// TIA Portal V20 export
FUNCTION_BLOCK "CallGlobal"   // FB48, LAD
TITLE = CallGlobal
// All blocks that provide data to the DB Global.Data are called here. That includes blocks to generate system data as well as blocks that connect handle multiple HMIs.
// stored: IsIECCheckEnabled true, MemoryReserve 100, SetENOAutomatically true
   VAR
      statClockSysMemOld { ExternalWritable := 'False'} : Byte;   // Old value system memory evaluation
      statTonTimer : Array[0..10] of IEC_TIMER;
      instLAF_PowerOnOff { ExternalWritable := 'False'} : "LAF_PowerOnOff";
      instLAF_HmiHeaderManager { ExternalWritable := 'False'} : "LAF_HmiHeaderManager";
      instLAF_ClockGen { ExternalWritable := 'False'} : "LAF_ClockGenerator";
      instLSNTP_Server { ExternalWritable := 'False'} : "LSNTP_Server";
      instRemoteAccess { ExternalWritable := 'False'} : "LRemoteAccess_MobilePanelMonitor";
      statPulse : Array[0..99] of Bool;
   END_VAR
   VAR_TEMP
      tempIndex : DInt;   // Temp variable for for loop
      tempAcknowledge : Bool;   // Summarized acknowledge command
      tempPowerOff : Bool;   // Summarized power off command
      tempPowerOn : Bool;   // Summarized power on command
      tempPowerStatus : Int;   // 0 - Off, 1 - Paused, 2 - On
      tempResultXor : Byte;   // Interim result of XOR operation
      tempPosPulse : Byte;   // Interim result puls calculation
   END_VAR
   VAR CONSTANT
      RESET_BUTTON__COULD_BE_ADDED_HERE : Bool := false;   // Placeholder for a potential global reset button
      TRUE : Bool := true;
   END_VAR
   VAR_TEMP   // added for the SCL form of the ladder/FBD networks
      _w1 : Bool;
      _w2 : Bool;
      _w3 : Bool;
   END_VAR
BEGIN

REGION Network 1 (SCL): Summarize HMI commands
   // Read commands for acknowledge, powerOn and powerOff from the different HMI panels and summarize them in temp variables for further logic in this block.
   // Initialize temp variables
   #tempAcknowledge :=
   #tempPowerOff :=
   #tempPowerOn := FALSE;

   // Loop through the HMI panels and summarize the commands
   FOR #tempIndex := 0 TO "NO_OF_PANELS" DO
       #tempAcknowledge := #tempAcknowledge OR "Hmi".mainHeader[#tempIndex].hmiToPlc.acknowledge;
       #tempPowerOff := #tempPowerOff OR "Hmi".mainHeader[#tempIndex].hmiToPlc.powerCommands.%X0;
       #tempPowerOn := #tempPowerOn OR "Hmi".mainHeader[#tempIndex].hmiToPlc.powerCommands.%X1;
   END_FOR;
END_REGION

REGION Network 2: Global Acknowledge
   // The global acknowledge command from the hmi button is assigned to Global.Data.general.acknowledge: This bit it forwarded to all underlaying modules
   // If a hard-wired global reset button exists, it can
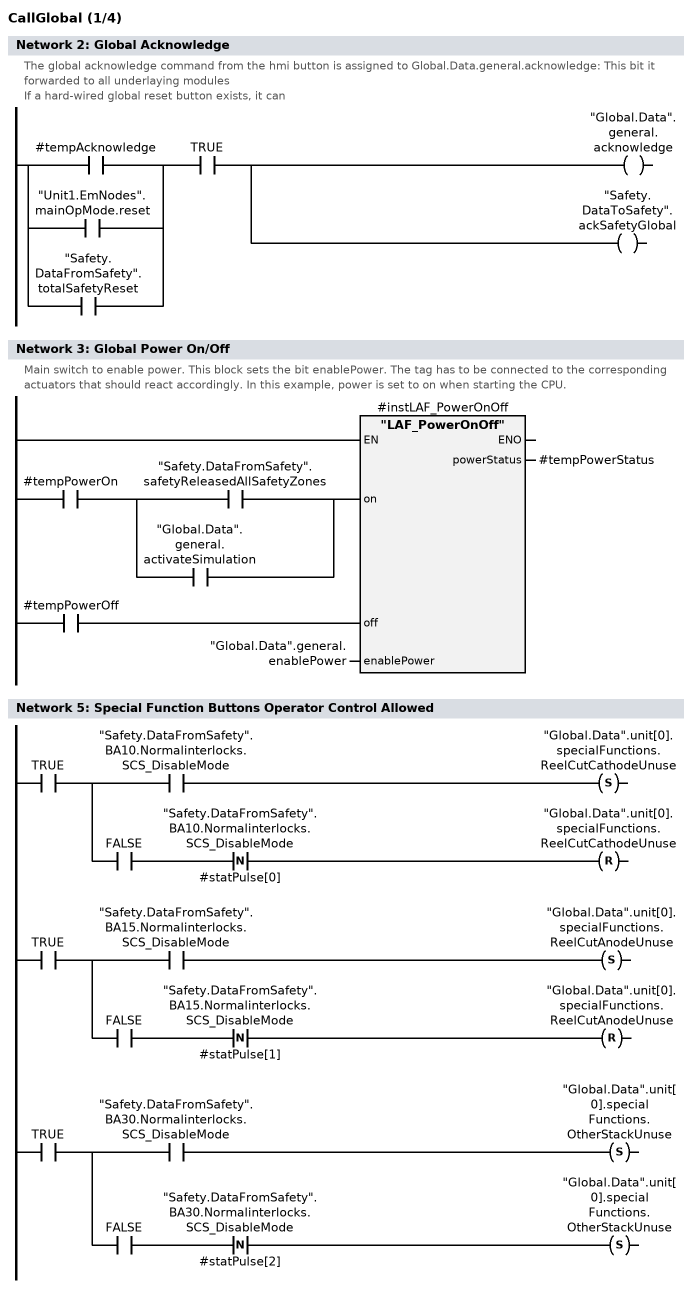
   RUNG wire#powerrail
      Contact( #tempAcknowledge )
      wire#w1
      Contact( TRUE )
      wire#w2
      Coil( "Global.Data".general.acknowledge )
   END_RUNG
   RUNG wire#powerrail
      Contact( "Unit1.EmNodes".mainOpMode.reset )
   END_RUNG wire#w1
   RUNG wire#powerrail
      Contact( "Safety.DataFromSafety".totalSafetyReset )
   END_RUNG wire#w1
   RUNG wire#w2
      Coil( "Safety.DataToSafety".ackSafetyGlobal )
   END_RUNG
   // the same network as SCL:
   "Global.Data".general.acknowledge := (#tempAcknowledge OR "Unit1.EmNodes".mainOpMode.reset OR "Safety.DataFromSafety".totalSafetyReset) AND TRUE;
   "Safety.DataToSafety".ackSafetyGlobal := "Global.Data".general.acknowledge;
END_REGION

REGION Network 3: Global Power On/Off
   // Main switch to enable power. This block sets the bit enablePower. The tag has to be connected to the corresponding actuators that should react accordingly. In this example, power is set to on when starting the CPU.
   RUNG wire#powerrail
      #instLAF_PowerOnOff(on := wire#w2, off := wire#w3, enablePower := "Global.Data".general.enablePower, powerStatus => #tempPowerStatus)
   END_RUNG
   RUNG wire#powerrail
      Contact( #tempPowerOn )
      wire#w1
      Contact( "Safety.DataFromSafety".safetyReleasedAllSafetyZones )
   END_RUNG wire#w2
   RUNG wire#w1
      Contact( "Global.Data".general.activateSimulation )
   END_RUNG wire#w2
   RUNG wire#powerrail
      Contact( #tempPowerOff )
   END_RUNG wire#w3
   // the same network as SCL:
   #instLAF_PowerOnOff(on := #tempPowerOn AND ("Safety.DataFromSafety".safetyReleasedAllSafetyZones OR "Global.Data".general.activateSimulation),   // "LAF_PowerOnOff"
                       off := #tempPowerOff,
                       enablePower := "Global.Data".general.enablePower,
                       powerStatus => #tempPowerStatus);
END_REGION

REGION Network 4 (SCL): Write power status to HMI panels
   // Write power status back to all connected HMI panels
   // Loop through the panels and set the power status
   FOR #tempIndex := 0 TO "NO_OF_PANELS" DO
       "Hmi".mainHeader[#tempIndex].plcToHmi.powerStatus := #tempPowerStatus;
   END_FOR;
END_REGION

REGION Network 5: Special Function Buttons Operator Control Allowed
   RUNG wire#powerrail
      Contact( TRUE )
      wire#w1
      Contact( "Safety.DataFromSafety".BA10.Normalinterlocks.SCS_DisableMode )
      S_Coil( "Global.Data".unit[0].specialFunctions.ReelCutCathodeUnuse )
   END_RUNG
   RUNG wire#w1
      Contact( FALSE )
      N_Contact(operand := "Safety.DataFromSafety".BA10.Normalinterlocks.SCS_DisableMode, bit := #statPulse[0])
      R_Coil( "Global.Data".unit[0].specialFunctions.ReelCutCathodeUnuse )
   END_RUNG
   RUNG wire#powerrail
      Contact( TRUE )
      wire#w2
      Contact( "Safety.DataFromSafety".BA15.Normalinterlocks.SCS_DisableMode )
      S_Coil( "Global.Data".unit[0].specialFunctions.ReelCutAnodeUnuse )
   END_RUNG
   RUNG wire#w2
      Contact( FALSE )
      N_Contact(operand := "Safety.DataFromSafety".BA15.Normalinterlocks.SCS_DisableMode, bit := #statPulse[1])
      R_Coil( "Global.Data".unit[0].specialFunctions.ReelCutAnodeUnuse )
   END_RUNG
   RUNG wire#powerrail
      Contact( TRUE )
      wire#w3
      Contact( "Safety.DataFromSafety".BA30.Normalinterlocks.SCS_DisableMode )
      S_Coil( "Global.Data".unit[0].specialFunctions.OtherStackUnuse )
   END_RUNG
   RUNG wire#w3
      Contact( FALSE )
      N_Contact(operand := "Safety.DataFromSafety".BA30.Normalinterlocks.SCS_DisableMode, bit := #statPulse[2])
      S_Coil( "Global.Data".unit[0].specialFunctions.OtherStackUnuse )
   END_RUNG
   // the same network as SCL:
   IF TRUE AND "Safety.DataFromSafety".BA10.Normalinterlocks.SCS_DisableMode THEN
       "Global.Data".unit[0].specialFunctions.ReelCutCathodeUnuse := TRUE;
   END_IF;
   #_w1 := TRUE AND FALSE AND NOT "Safety.DataFromSafety".BA10.Normalinterlocks.SCS_DisableMode AND #statPulse[0];   // falling edge of "Safety.DataFromSafety".BA10.Normalinterlocks.SCS_DisableMode
   #statPulse[0] := "Safety.DataFromSafety".BA10.Normalinterlocks.SCS_DisableMode;
   IF #_w1 THEN "Global.Data".unit[0].specialFunctions.ReelCutCathodeUnuse := FALSE; END_IF;
   IF TRUE AND "Safety.DataFromSafety".BA15.Normalinterlocks.SCS_DisableMode THEN
       "Global.Data".unit[0].specialFunctions.ReelCutAnodeUnuse := TRUE;
   END_IF;
   #_w2 := TRUE AND FALSE AND NOT "Safety.DataFromSafety".BA15.Normalinterlocks.SCS_DisableMode AND #statPulse[1];   // falling edge of "Safety.DataFromSafety".BA15.Normalinterlocks.SCS_DisableMode
   #statPulse[1] := "Safety.DataFromSafety".BA15.Normalinterlocks.SCS_DisableMode;
   IF #_w2 THEN "Global.Data".unit[0].specialFunctions.ReelCutAnodeUnuse := FALSE; END_IF;
   IF TRUE AND "Safety.DataFromSafety".BA30.Normalinterlocks.SCS_DisableMode THEN
       "Global.Data".unit[0].specialFunctions.OtherStackUnuse := TRUE;
   END_IF;
   #_w3 := TRUE AND FALSE AND NOT "Safety.DataFromSafety".BA30.Normalinterlocks.SCS_DisableMode AND #statPulse[2];   // falling edge of "Safety.DataFromSafety".BA30.Normalinterlocks.SCS_DisableMode
   #statPulse[2] := "Safety.DataFromSafety".BA30.Normalinterlocks.SCS_DisableMode;
   IF #_w3 THEN "Global.Data".unit[0].specialFunctions.OtherStackUnuse := TRUE; END_IF;
END_REGION

REGION Network 6: HMI Control Header
   // Read the input from the control header in the HMI an distribute information to the according units. Vice versa, summarize the unit information and provide it to the control header to display e.g. the modes and states.
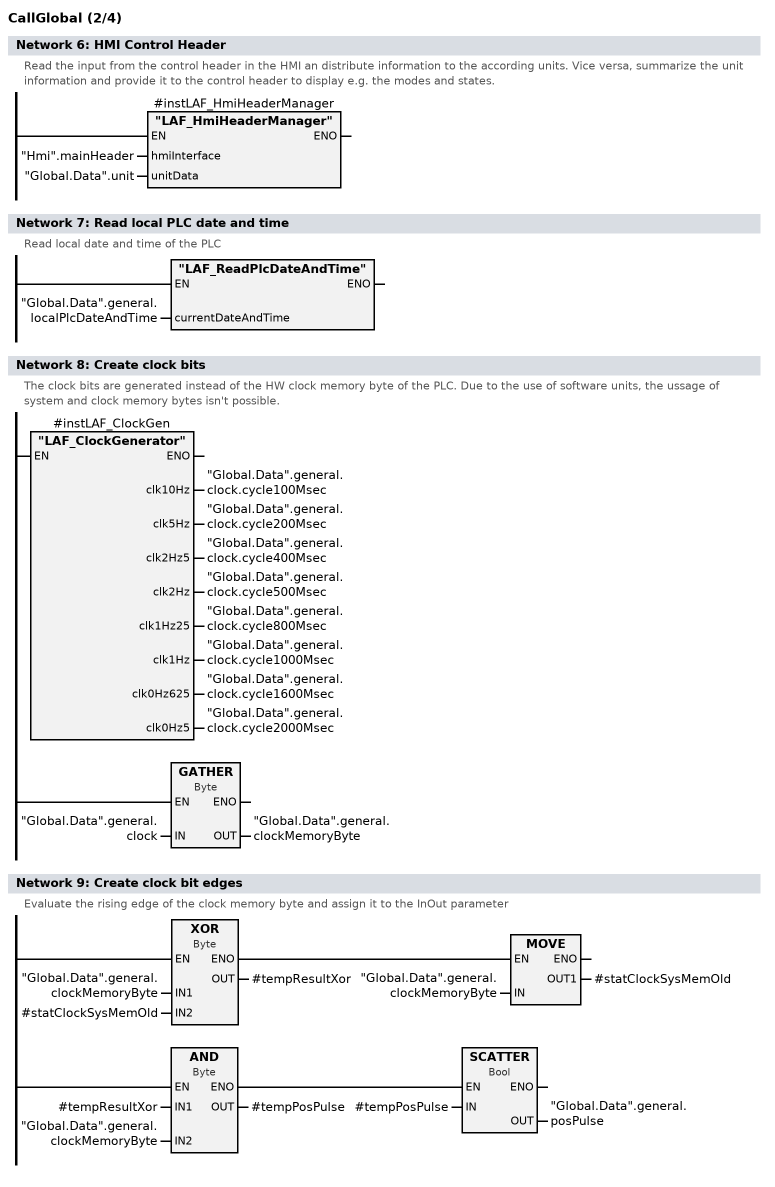
   RUNG wire#powerrail
      #instLAF_HmiHeaderManager(hmiInterface := "Hmi".mainHeader, unitData := "Global.Data".unit)
   END_RUNG
   // the same network as SCL:
   #instLAF_HmiHeaderManager(hmiInterface := "Hmi".mainHeader, unitData := "Global.Data".unit);   // "LAF_HmiHeaderManager"
END_REGION

REGION Network 7: Read local PLC date and time
   // Read local date and time of the PLC
   RUNG wire#powerrail
      "LAF_ReadPlcDateAndTime"(currentDateAndTime := "Global.Data".general.localPlcDateAndTime)
   END_RUNG
   // the same network as SCL:
   "LAF_ReadPlcDateAndTime"(currentDateAndTime := "Global.Data".general.localPlcDateAndTime);
END_REGION

REGION Network 8: Create clock bits
   // The clock bits are generated instead of the HW clock memory byte of the PLC. Due to the use of software units, the ussage of system and clock memory bytes isn't possible.
   RUNG wire#powerrail
      #instLAF_ClockGen(clk10Hz => "Global.Data".general.clock.cycle100Msec, clk5Hz => "Global.Data".general.clock.cycle200Msec, clk2Hz5 => "Global.Data".general.clock.cycle400Msec, clk2Hz => "Global.Data".general.clock.cycle500Msec, clk1Hz25 => "Global.Data".general.clock.cycle800Msec, clk1Hz => "Global.Data".general.clock.cycle1000Msec, clk0Hz625 => "Global.Data".general.clock.cycle1600Msec, clk0Hz5 => "Global.Data".general.clock.cycle2000Msec)
   END_RUNG
   RUNG wire#powerrail
      { S7_Templates := "[dest_type := Byte, src_type := Bool]" } GATHER(IN := "Global.Data".general.clock, OUT => "Global.Data".general.clockMemoryByte)
   END_RUNG
   // the same network as SCL:
   #instLAF_ClockGen(clk10Hz => "Global.Data".general.clock.cycle100Msec,   // "LAF_ClockGenerator"
                     clk5Hz => "Global.Data".general.clock.cycle200Msec,
                     clk2Hz5 => "Global.Data".general.clock.cycle400Msec,
                     clk2Hz => "Global.Data".general.clock.cycle500Msec,
                     clk1Hz25 => "Global.Data".general.clock.cycle800Msec,
                     clk1Hz => "Global.Data".general.clock.cycle1000Msec,
                     clk0Hz625 => "Global.Data".general.clock.cycle1600Msec,
                     clk0Hz5 => "Global.Data".general.clock.cycle2000Msec);
   GATHER(IN := "Global.Data".general.clock, OUT => "Global.Data".general.clockMemoryByte);
END_REGION

REGION Network 9: Create clock bit edges
   // Evaluate the rising edge of the clock memory byte and assign it to the InOut parameter
   #tempResultXor := "Global.Data".general.clockMemoryByte XOR #statClockSysMemOld;
   #statClockSysMemOld := "Global.Data".general.clockMemoryByte;
   #tempPosPulse := #tempResultXor AND "Global.Data".general.clockMemoryByte;
   SCATTER(IN := #tempPosPulse, OUT => "Global.Data".general.posPulse);
END_REGION

REGION Network 10: Time Synchronisation (NTP)
   // With the LSNTP_Server block, the NTP server will be enabled on S7 PLC, to wich the NTP client (e.g. Panel), can synchronize their data and time.
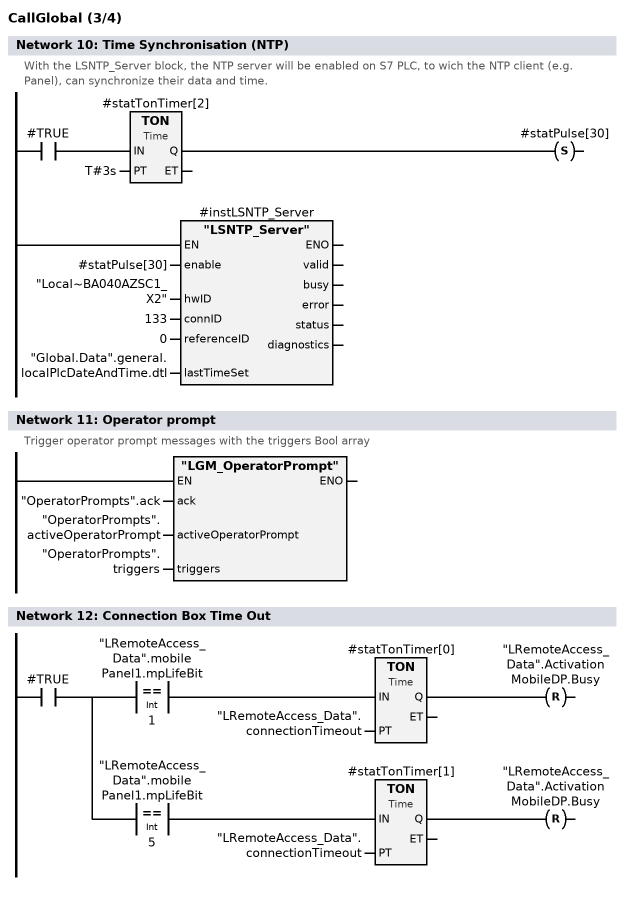
   RUNG wire#powerrail
      Contact( #TRUE )
      { S7_Templates := "time_type := Time" } #statTonTimer[2].TON(pt := T#3s, et =>)
      S_Coil( #statPulse[30] )
   END_RUNG
   RUNG wire#powerrail
      #instLSNTP_Server(enable := #statPulse[30], hwID := "Local~BA040AZSC1_X2", connID := 133, referenceID := 0, lastTimeSet := "Global.Data".general.localPlcDateAndTime.dtl, valid =>, busy =>, error =>, status =>, diagnostics =>)
   END_RUNG
   // the same network as SCL:
   #statTonTimer[2].TON(IN := #TRUE, PT := T#3s);
   IF #statTonTimer[2].Q THEN #statPulse[30] := TRUE; END_IF;
   #instLSNTP_Server(enable := #statPulse[30],   // "LSNTP_Server"
                     hwID := "Local~BA040AZSC1_X2",
                     connID := 133,
                     referenceID := 0,
                     lastTimeSet := "Global.Data".general.localPlcDateAndTime.dtl);
END_REGION

REGION Network 11: Operator prompt
   // Trigger operator prompt messages with the triggers Bool array
   RUNG wire#powerrail
      "LGM_OperatorPrompt"(ack := "OperatorPrompts".ack, activeOperatorPrompt := "OperatorPrompts".activeOperatorPrompt, triggers := "OperatorPrompts".triggers)
   END_RUNG
   // the same network as SCL:
   "LGM_OperatorPrompt"(ack := "OperatorPrompts".ack,
                        activeOperatorPrompt := "OperatorPrompts".activeOperatorPrompt,
                        triggers := "OperatorPrompts".triggers);
END_REGION

REGION Network 12: Connection Box Time Out
   RUNG wire#powerrail
      Contact( #TRUE )
      wire#w1
      { S7_Templates := "SrcType := Int" } EQ_Contact(in1 := "LRemoteAccess_Data".mobilePanel1.mpLifeBit, in2 := 1)
      { S7_Templates := "time_type := Time" } #statTonTimer[0].TON(pt := "LRemoteAccess_Data".connectionTimeout, et =>)
      R_Coil( "LRemoteAccess_Data".ActivationMobileDP.Busy )
   END_RUNG
   RUNG wire#w1
      { S7_Templates := "SrcType := Int" } EQ_Contact(in1 := "LRemoteAccess_Data".mobilePanel1.mpLifeBit, in2 := 5)
      { S7_Templates := "time_type := Time" } #statTonTimer[1].TON(pt := "LRemoteAccess_Data".connectionTimeout, et =>)
      R_Coil( "LRemoteAccess_Data".ActivationMobileDP.Busy )
   END_RUNG
   // the same network as SCL:
   #statTonTimer[0].TON(IN := #TRUE AND ("LRemoteAccess_Data".mobilePanel1.mpLifeBit = 1),
                        PT := "LRemoteAccess_Data".connectionTimeout);
   IF #statTonTimer[0].Q THEN "LRemoteAccess_Data".ActivationMobileDP.Busy := FALSE; END_IF;
   #statTonTimer[1].TON(IN := #TRUE AND ("LRemoteAccess_Data".mobilePanel1.mpLifeBit = 5),
                        PT := "LRemoteAccess_Data".connectionTimeout);
   IF #statTonTimer[1].Q THEN "LRemoteAccess_Data".ActivationMobileDP.Busy := FALSE; END_IF;
END_REGION

REGION Network 13: Connection box is connected
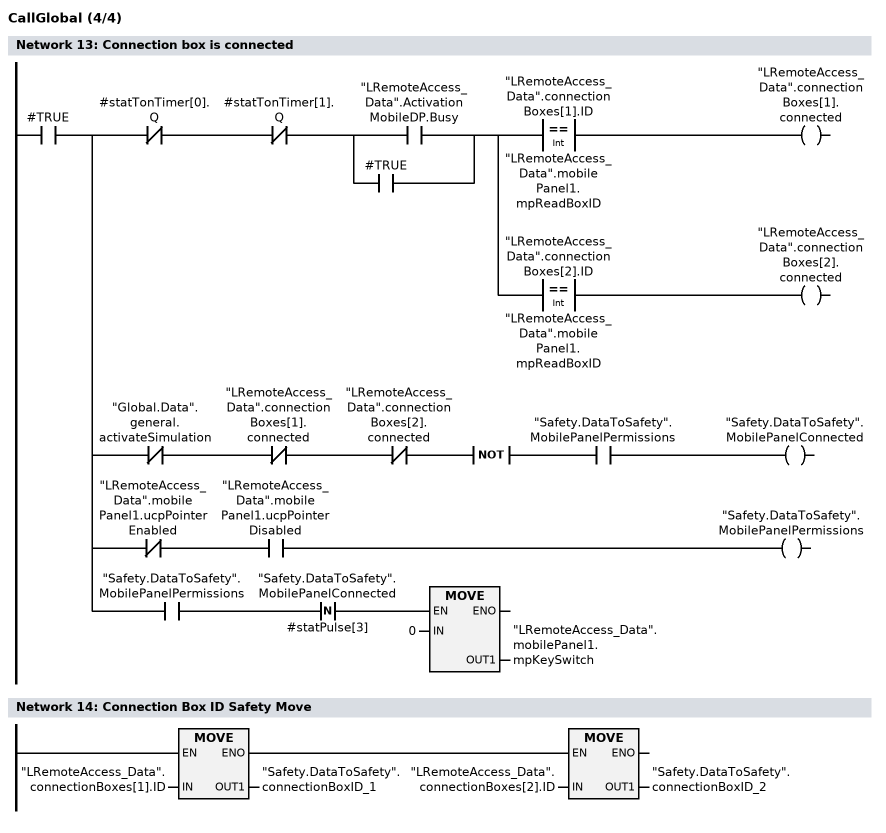
   RUNG wire#powerrail
      Contact( #TRUE )
      wire#w1
      I_Contact( #statTonTimer[0].Q )
      I_Contact( #statTonTimer[1].Q )
      wire#w2
      Contact( "LRemoteAccess_Data".ActivationMobileDP.Busy )
      wire#w3
      { S7_Templates := "SrcType := Int" } EQ_Contact(in1 := "LRemoteAccess_Data".connectionBoxes[1].ID, in2 := "LRemoteAccess_Data".mobilePanel1.mpReadBoxID)
      Coil( "LRemoteAccess_Data".connectionBoxes[1].connected )
   END_RUNG
   RUNG wire#w2
      Contact( #TRUE )
   END_RUNG wire#w3
   RUNG wire#w3
      { S7_Templates := "SrcType := Int" } EQ_Contact(in1 := "LRemoteAccess_Data".connectionBoxes[2].ID, in2 := "LRemoteAccess_Data".mobilePanel1.mpReadBoxID)
      Coil( "LRemoteAccess_Data".connectionBoxes[2].connected )
   END_RUNG
   RUNG wire#w1
      I_Contact( "Global.Data".general.activateSimulation )
      I_Contact( "LRemoteAccess_Data".connectionBoxes[1].connected )
      I_Contact( "LRemoteAccess_Data".connectionBoxes[2].connected )
      Not()
      Contact( "Safety.DataToSafety".MobilePanelPermissions )
      Coil( "Safety.DataToSafety".MobilePanelConnected )
   END_RUNG
   RUNG wire#w1
      I_Contact( "LRemoteAccess_Data".mobilePanel1.ucpPointerEnabled )
      Contact( "LRemoteAccess_Data".mobilePanel1.ucpPointerDisabled )
      Coil( "Safety.DataToSafety".MobilePanelPermissions )
   END_RUNG
   RUNG wire#w1
      Contact( "Safety.DataToSafety".MobilePanelPermissions )
      N_Contact(operand := "Safety.DataToSafety".MobilePanelConnected, bit := #statPulse[3])
      Move(in := 0, out1 => "LRemoteAccess_Data".mobilePanel1.mpKeySwitch)
   END_RUNG
   // the same network as SCL:
   #_w1 := #TRUE AND NOT #statTonTimer[0].Q AND NOT #statTonTimer[1].Q AND ("LRemoteAccess_Data".ActivationMobileDP.Busy OR #TRUE);
   "LRemoteAccess_Data".connectionBoxes[1].connected := #_w1 AND ("LRemoteAccess_Data".connectionBoxes[1].ID = "LRemoteAccess_Data".mobilePanel1.mpReadBoxID);
   "LRemoteAccess_Data".connectionBoxes[2].connected := #_w1 AND ("LRemoteAccess_Data".connectionBoxes[2].ID = "LRemoteAccess_Data".mobilePanel1.mpReadBoxID);
   "Safety.DataToSafety".MobilePanelConnected := NOT (#TRUE AND NOT "Global.Data".general.activateSimulation AND NOT "LRemoteAccess_Data".connectionBoxes[1].connected AND NOT "LRemoteAccess_Data".connectionBoxes[2].connected) AND "Safety.DataToSafety".MobilePanelPermissions;
   "Safety.DataToSafety".MobilePanelPermissions := #TRUE AND NOT "LRemoteAccess_Data".mobilePanel1.ucpPointerEnabled AND "LRemoteAccess_Data".mobilePanel1.ucpPointerDisabled;
   #_w2 := #TRUE AND "Safety.DataToSafety".MobilePanelPermissions AND NOT "Safety.DataToSafety".MobilePanelConnected AND #statPulse[3];   // falling edge of "Safety.DataToSafety".MobilePanelConnected
   #statPulse[3] := "Safety.DataToSafety".MobilePanelConnected;
   IF #_w2 THEN "LRemoteAccess_Data".mobilePanel1.mpKeySwitch := 0; END_IF;
END_REGION

REGION Network 14: Connection Box ID Safety Move
   RUNG wire#powerrail
      Move(in := "LRemoteAccess_Data".connectionBoxes[1].ID, out1 => "Safety.DataToSafety".connectionBoxID_1)
      Move(in := "LRemoteAccess_Data".connectionBoxes[2].ID, out1 => "Safety.DataToSafety".connectionBoxID_2)
   END_RUNG
   // the same network as SCL:
   "Safety.DataToSafety".connectionBoxID_1 := "LRemoteAccess_Data".connectionBoxes[1].ID;
   "Safety.DataToSafety".connectionBoxID_2 := "LRemoteAccess_Data".connectionBoxes[2].ID;
END_REGION
END_FUNCTION_BLOCK
